(* IEC 61131-3 sources: plc_generation_empirical_study/datasets/_archive/native_profile_v5_20260810/tasks/C04_M01_falling_edge_pulse, 2 files *)

(* ---- interface.st ---- *)
FUNCTION_BLOCK C04_M01_falling_edge_pulse
VAR_INPUT
    Signal : BOOL;
    Arm : BOOL;
END_VAR
VAR_OUTPUT
    Pulse : BOOL;
    Armed : BOOL;
END_VAR
END_FUNCTION_BLOCK

(* ---- reference.st ---- *)
FUNCTION_BLOCK C04_M01_falling_edge_pulse
VAR_INPUT
    Signal : BOOL;
    Arm : BOOL;
END_VAR
VAR_OUTPUT
    Pulse : BOOL;
    Armed : BOOL;
END_VAR
VAR
    PrevSignal : BOOL := FALSE;
END_VAR

Pulse := Arm AND (NOT Signal) AND PrevSignal;
Armed := Arm;
PrevSignal := Signal;

END_FUNCTION_BLOCK
